FUNCTION_BLOCK Signal_OR (* Basic Function Block Type *)
  (* Standard: 61499-2 *)
  (* Version 0.0, 2/8/2018, Eskimos, nxtControl GmbH, Template *)
  PACKAGE Main;
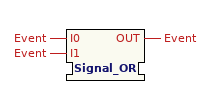
  EVENT_INPUT
    I0; (* Initialization Request *)
    I1; (* Normal Execution Request *)
  END_EVENT
  EVENT_OUTPUT
    OUT; (* Initialization Confirm *)
  END_EVENT
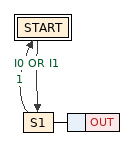
  EC_STATES
    START; (* Initial State *)
    S1 : -> OUT; (* Normal execution *)
  END_STATES
  EC_TRANSITIONS
    START TO S1 := I0 OR I1;
    S1 TO START := 1;
  END_TRANSITIONS
END_FUNCTION_BLOCK
